// Checks if the given generic value represents a real (floating-point) number type.
FUNCTION F_IsRealNumberGeneric : BOOL // TRUE if the generic value represents a real (floating-point) number type.
VAR_INPUT
	Value : FsCommon.T_Generic; // The generic value to check.
END_VAR

F_IsRealNumberGeneric := 
	Value.TypeClass = __SYSTEM.TYPE_CLASS.TYPE_REAL
	OR
	Value.TypeClass = __SYSTEM.TYPE_CLASS.TYPE_LREAL;

END_FUNCTION

(* stored: Version 1.1.0.1
   POU F_IsRealNumberGeneric: Id {1aad7acb-a07f-07d5-30aa-0646f52e840e}, SpecialFunc None *)
